TYPE ST_GC_ServiceCtrl :
STRUCT
	SpinAxisJog : ST_GCSpinAxisJogCtrl;
	SpinAxisMoveAbs : ST_GCSpinAxisMoveAbsCtrl;
	SpinAxisMoveVel	: ST_GCSpinAxisMoveVelCtrl;
END_STRUCT
END_TYPE

(* stored: Version 1.1.0.1, ProductVersion 3.1.4026.18
   DUT ST_GC_ServiceCtrl: Id {ffd8beff-04a4-4f84-92ab-5776cc33b725} *)
